Fanuc TP program (LS listing): TITAN4.ls

/PROG TITAN4
/ATTR
/MN

: ! This is the blast program for a Titan 4 container ;

: UFRAME_NUM=1 ;
: UTOOL_NUM=1 ;

: CALL TITAN4_INIT ;
: CALL HOME ;
: CALL TITAN4_EAST_OUT ;


/POS
/END
